{attribute 'GeneratedUsingTerminal: EP5101-2011-0016'}
{attribute addProperty BoxType "EP5101-2011-0016"}
{attribute addProperty Id "StatusAT %I*Status_E2E79E8513Counter_valueAT %I*UINT2Latch_valueAT %I*UINT2"}
{attribute addProperty CRC "1100541755"}
{attribute addProperty Size "17"}
TYPE ENC_Status_compact_4198EF3B :
STRUCT
	{attribute addProperty Name "Status"}
	Status AT %I* : Status_E2E79E85;
	{attribute addProperty Name "Counter_value"}
	Counter_value AT %I* : UINT;
	{attribute addProperty Name "Latch_value"}
	Latch_value AT %I* : UINT;
END_STRUCT
END_TYPE

(* stored: Version 1.2.0.0, ProductVersion 3.1.4024.9
   DUT ENC_Status_compact_4198EF3B: Id {37e5ed38-1665-4dfa-973d-aa8ea7df6a44} *)
